// TIA Portal V19 export
FUNCTION "TEST TEMPERATURE" : Void   // FC18, STL
TITLE = TEST TEMPERATURES
{ S7_Optimized_Access := 'TRUE' }
NAME : TESTTEMP
VERSION : 0.0
// Comment
// stored: AutoNumber false
BEGIN

NETWORK
TITLE = TEST TEMPERATURES
      AN    "TEST TEMPS. PRESTERILI";
      JC    M001;
      O(;
      L     "MeasuredValues".TT0176REAL;  //"DB-ANALOG INPUT".TT0176MEAS
      L     "Setpoints".TT0176MinTempUnster;  //"DB SETPOINTS".TT0176MinTempUnster
      <R;
      S     "ProcessAndPbAlarms"."A"[33];  //A33_TT0176TooLow// 0176 too low
      );
      O(;
      L     "MeasuredValues".TT0160REAL;  //"DB-ANALOG INPUT".TT0160MEAS
      L     "Setpoints".TT0160MinTempUnster;  //"DB SETPOINTS".TT0160MinTempUnster
      <R;
      S     "ProcessAndPbAlarms"."A"[34];  //A34_TT0160TooLow// 0160 too low
      );
      O(;
      L     "MeasuredValues".TT0163REAL;  // "DB-ANALOG INPUT".TT0163MEAS
      L     "Setpoints".TT0163MinTempUnster;  //"DB SETPOINTS".TT0163MinTempUnster
      <R;
      S     "ProcessAndPbAlarms"."A"[35];  //A35_TT0163TooLow// 0163 too low
      );
      O(;
      L     "MeasuredValues".TT0178REAL;  // "DB-ANALOG INPUT".TT0178MEAS
      L     "Setpoints".TT0178MinTempUnster;  //"DB SETPOINTS".TT0178MinTempUnster
      <R;
      S     "ProcessAndPbAlarms"."A"[36];  //A36_TT0178TooLow// 0178 too low
      );
      O(;
      L     "MeasuredValues".TT0951REAL;  // "DB-ANALOG INPUT".TT0951MEAS
      L     "Setpoints_Hamba".TT0951StartSterileTime;  //"DB SETPOINTS".TT0951MinTempUnster
      <R;
      S     "ProcessAndPbAlarms"."A"[57];  //A57_TT0951TooLow// 0951 too low
      );
      O(;
      L     "IF_Device".TTX_09_30.ProcessData.Temperature;
      L     "SetpointsV0101Condensate".TT0930_Low_Prod;
      <R;
      S     "ProcessAndPbAlarms"."A"[66];  //A66_TT0930_Low_SIP// 0951 too low
      );
      R     "T 14 STERILE TIME";
      R     "S3 PRESTERILIZING";
      R     "TEST TEMPS. PRESTERILI";
      R     "M_Barrier_Sterlising";
      BEU;
M001: NOP   0;

NETWORK
TITLE = ProcessAlarm
      AN    "TEST BARRIERS";
      R     "ProcessAndPbAlarms"."A"[37];  //A37_TT0176Low// 0176 low
      R     "DUMMY TEST TT 01.76";
      R     "ProcessAndPbAlarms"."A"[38];  //A38_TT0178Low// 0178 low
      R     "DUMMY TEST TT 01.78";
      R     "ProcessAndPbAlarms"."A"[58];  //A58_TT0951Low// 0951 low
      R     "DUMMY TEST TT 09.51";
      BEC;

NETWORK
TITLE = DUMMY TEST TT 01.76 AS BARRIER
      AN    "MY0147";
      JC    M002;
      A     "MY0113";
      JC    M002;
      L     "MeasuredValues".TT0176REAL;  // "DB-ANALOG INPUT".TT0176MEAS
      L     "Setpoints".TT0176LowTemp;  //"DB SETPOINTS".TT0176LowTemp
      >R;
      JC    M002;
      A     "DUMMY TEST TT 01.76";
      JC    M003;
      S     "DUMMY TEST TT 01.76";
      S     "TIM36";
      JU    END;
M003: A     "T 36 DELAY TT 01.76";
      JC    END;
      S     "ProcessAndPbAlarms"."A"[37];  //A37_TT0176Low// 0176 low
      JU    END;
M002: R     "ProcessAndPbAlarms"."A"[37];  //A37_TT0176Low// 0176 low
      R     "DUMMY TEST TT 01.76";
END:  NOP   0;

NETWORK
TITLE = DUMMY TEST TT 01.78 AS BARRIER
      A     "MY0108";
      JC    c001;
      L     "MeasuredValues".TT0178REAL;  // "DB-ANALOG INPUT".TT0178MEAS
      L     "Setpoints".TT0178LowTemp;  //"DB SETPOINTS".TT0178LowTemp
      >R;
      JC    c001;
      A     "DUMMY TEST TT 01.78";
      JC    c002;
      S     "DUMMY TEST TT 01.78";
      S     "TIM37";
      JU    c003;
c002: A     "T 37 DELAY TT 01.78";
      JC    c003;
      S     "ProcessAndPbAlarms"."A"[38];  //A38_TT0178Low// 0178 low
      JU    c003;
c001: R     "ProcessAndPbAlarms"."A"[38];  //A38_TT0178Low// 0178 low
      R     "DUMMY TEST TT 01.78";
c003: NOP   0;

NETWORK
TITLE = DUMMY TEST TT 09.51 AS BARRIER
      CLR;
      A     "DisableMonitoringTT0951";
      JC    x003;

      L     "MeasuredValues".TT0951REAL;  // "DB-ANALOG INPUT".TT0951MEAS
      L     "Setpoints_Hamba".TT0951BarrierTemp;  //"DB SETPOINTS".TT0951LowTemp
      >R;
      JC    x001;
      A     "DUMMY TEST TT 09.51";
      JC    x002;
      S     "DUMMY TEST TT 09.51";
      S     "TIM56";  // TT0951BarrierTime
      JU    x003;
x002: A     "Tag_55";
      JC    x003;
      S     "ProcessAndPbAlarms"."A"[58];  //A58_TT0951Low// 0951 low
      R     "M_Barrier_Sterlising";
      JU    x003;
x001: R     "ProcessAndPbAlarms"."A"[58];  //A58_TT0951Low// 0951 low
      R     "DUMMY TEST TT 09.51";
x003: NOP   0;
END_FUNCTION
